      A     #s_Status.THO_400VAC_GRP16;
      =     #o_ST_THO_400Vac_GRP16;

      A     #s_Status.THO_230VAC_GRP01;
      =     #o_ST_THO_230Vac_GRP01;

      A     #s_Status.THO_230VAC_GRP02;
      =     #o_ST_THO_230Vac_GRP02;

      A     #s_Status.THO_230VAC_GRP03;
      =     #o_ST_THO_230Vac_GRP03;

      A     #s_Status.THO_230VAC_GRP04;
      =     #o_ST_THO_230Vac_GRP04;

      A     #s_Status.THO_230VAC_GRP05;
      =     #o_ST_THO_230Vac_GRP05;

      A     #s_Status.THO_230VAC_GRP06;
      =     #o_ST_THO_230Vac_GRP06;

      A     #s_Status.THO_230VAC_GRP07;
      =     #o_ST_THO_230Vac_GRP07;

      A     #s_Status.THO_230VAC_GRP08;
      =     #o_ST_THO_230Vac_GRP08;

      A     #s_Status.THO_230VAC_GRP09;
      =     #o_ST_THO_230Vac_GRP09;

      A     #s_Status.THO_230VAC_GRP10;
      =     #o_ST_THO_230Vac_GRP10;

      A     #s_Status.THO_230VAC_GRP11;
      =     #o_ST_THO_230Vac_GRP11;

      A     #s_Status.THO_230VAC_GRP12;
      =     #o_ST_THO_230Vac_GRP12;

      A     #s_Status.THO_230VAC_GRP13;
      =     #o_ST_THO_230Vac_GRP13;

      A     #s_Status.THO_230VAC_GRP14;
      =     #o_ST_THO_230Vac_GRP14;

      A     #s_Status.THO_230VAC_GRP15;
      =     #o_ST_THO_230Vac_GRP15;

      A     #s_Status.THO_230VAC_GRP16;
      =     #o_ST_THO_230Vac_GRP16;

      A     #s_Status.No_Power_GRP01;
      =     #o_ST_No_Power_GRP01;

      A     #s_Status.No_Power_GRP02;
      =     #o_ST_No_Power_GRP02;

      A     #s_Status.No_Power_GRP03;
      =     #o_ST_No_Power_GRP03;

      A     #s_Status.No_Power_GRP04;
      =     #o_ST_No_Power_GRP04;

      A     #s_Status.No_Power_GRP05;
      =     #o_ST_No_Power_GRP05;

      A     #s_Status.No_Power_GRP06;
      =     #o_ST_No_Power_GRP06;

      A     #s_Status.No_Power_GRP07;
      =     #o_ST_No_Power_GRP07;

      A     #s_Status.No_Power_GRP08;
      =     #o_ST_No_Power_GRP08;

      A     #s_Status.No_Power_GRP09;
      =     #o_ST_No_Power_GRP09;

      A     #s_Status.No_Power_GRP10;
      =     #o_ST_No_Power_GRP10;

      A     #s_Status.No_Power_GRP11;
      =     #o_ST_No_Power_GRP11;

      A     #s_Status.No_Power_GRP12;
      =     #o_ST_No_Power_GRP12;

      A     #s_Status.No_Power_GRP13;
      =     #o_ST_No_Power_GRP13;

      A     #s_Status.No_Power_GRP14;
      =     #o_ST_No_Power_GRP14;

      A     #s_Status.No_Power_GRP15;
      =     #o_ST_No_Power_GRP15;

      A     #s_Status.No_Power_GRP16;
      =     #o_ST_No_Power_GRP16;

      A     #s_Status.PN1_Error;
      =     #o_ST_PN1_Err;

      A     #s_Status.PN1_NotPrsnt;
      =     #o_ST_PN1_NotPrsnt;

      A     #s_Status.PN2_Error;
      =     #o_ST_PN2_Err;

      A     #s_Status.PN2_NotPrsnt;
      =     #o_ST_PN2_NotPrsnt;

      A     #s_Status.PN3_Error;
      =     #o_ST_PN3_Err;

      A     #s_Status.PN3_NotPrsnt;
      =     #o_ST_PN3_NotPrsnt;

END_FUNCTION_BLOCK

